FUNCTION_BLOCK FB_CleaningProcessStateCappingExit EXTENDS FB_CleaningProcessStateBase
VAR_INPUT
END_VAR

VAR_OUTPUT
END_VAR

VAR
END_VAR

METHOD mCleaningOp : BOOL
VAR_INPUT
	sI_Operation : EN_CLEANING_OP;
END_VAR
//Set mode and start process when successful
(*HOA TEST
IF NOT bL_DevOpActive THEN
  bL_DevOpActive := I_ParentCallback.mSetMode(sI_Operation);
  mCleaningOp    := TRUE; //report success
END_IF*) mCleaningOp    := TRUE;

//Switch to production mode if no operation active
IF I_MachineStatus.pSafetyOk AND I_MachineStatus.pMachineReady AND NOT bL_DevOpActive THEN
  IF sI_Operation = eOPCAPENTER THEN
    I_ParentCallback.mChangeState(EN_Cleaning_State.Capping);
  ELSIF sI_Operation = eOPCAPEXIT THEN
    I_ParentCallback.mChangeState(EN_Cleaning_State.CappingExit);
  ELSIF sI_Operation = eOPCLEAN THEN
    I_ParentCallback.mChangeState(EN_Cleaning_State.Cleaning);
  ELSIF sI_Operation = eOPPURGE THEN
    I_ParentCallback.mChangeState(EN_Cleaning_State.Capping);
  END_IF
END_IF
END_METHOD

METHOD mEntryAction
VAR_INPUT
END_VAR
iL_CurrentStep := 0;

// Launch initial command to bring system to service mode
bL_DevOpActive := I_ParentCallback.mSetMode(EN_CLEANING_OP.eOPCAPEXIT);
END_METHOD

METHOD mProduction : BOOL
VAR_INPUT
END_VAR
//Switch to production mode if no operation active
IF I_MachineStatus.pSafetyOk AND I_MachineStatus.pMachineReady AND NOT bL_DevOpActive THEN
	I_ParentCallback.mChangeState(EN_Cleaning_State.Production);
END_IF
END_METHOD

METHOD mService : BOOL
VAR_INPUT
END_VAR
//Switch to service mode
IF NOT bL_DevOpActive THEN
	I_ParentCallback.mChangeState(EN_Cleaning_State.Service);
END_IF
END_METHOD

METHOD mStateAction
VAR_INPUT
END_VAR

VAR
	sL_DeviceStatus: ST_CLEANING_DEV_STATUS;
END_VAR
sL_DeviceStatus := I_ParentCallback.pDeviceStatus;
SUPER^.pInitDone := TRUE;

IF bL_DevOpActive THEN
	mDevOp();	
END_IF



//If error go to error mode
IF sL_DeviceStatus.bError THEN
	I_ParentCallback.mChangeState(EN_Cleaning_State.Error);
END_IF
END_METHOD

END_FUNCTION_BLOCK

(* stored: Version 1.1.0.1, ProductVersion 3.1.4024.11
   POU FB_CleaningProcessStateCappingExit: Id {69b936a6-3f6e-42db-974b-ab15d00ff0c1}, SpecialFunc None
   Method mCleaningOp: Id {95578ed7-8f88-4cda-9c10-b1850dfe31d4}
   Method mEntryAction: Id {ea1c4cf2-16ff-41f2-a834-5ad83c17d1f9}
   Method mProduction: Id {226b6699-13e2-4d66-a737-d6e5f00d6356}
   Method mService: Id {f707c4cb-7610-456a-88bd-31f2d9af3c4e}
   Method mStateAction: Id {581c1da2-f00b-4d3a-9714-3ac09c6e32fd} *)
